// TwinCAT 3 PLC project PLC_Project
// ProgramVersion: 3.1.4024.0
// libraries:
//   Tc2_Standard, * (Beckhoff Automation GmbH)
//   Tc2_System, * (Beckhoff Automation GmbH)
//   Tc3_Module, * (Beckhoff Automation GmbH)
//   VisuDialogs, * (System)
//   VisuSymbols,3.5.10.0,System
// project tree:
//   / GlobalTextList.TcGTLO, PlcTask.TcTTO
//   GVLs/ GVL_Analogue_Transducer_Instruments.TcGVL, GVL_Analogue_Transducer_Instruments_IO_Addresses.TcGVL
//   POUs/ Analogue_Processing.TcPOU, MAIN.TcPOU
//   POUs/Function Blocks/ Sensor_Calibration_Multipoint.TcPOU, Temperature_Transducer.TcPOU
//   VISUs/ VisualizationManager.TcVMO (not stored), Visualization_Calibration_Screen.TcVIS
// real-time tasks:
//   TASK PlcTask: cycle T#10ms, priority 20, ADS port 350
// I/O:
//   DEVICE Device 1 (EtherCAT) (disabled), AmsNetId 10.0.2.15.2.1
//     Term 1 (EK1101) [EK1101 EtherCAT Coupler (2A E-Bus, ID switch)]
//       Term 2 (EL3202-0020) [EL3202-0020 2Ch. Ana. Input PT100 (RTD), High Precision, calibrated]
// variable links:
//   PLC Project/PLC Project Instance <-> Device 1 (EtherCAT)/Term 1 (EK1101)/Term 2 (EL3202-0020)
//     PlcTask Inputs/GVL_Analogue_Transducer_Instruments_IO_Addresses.Temperature_Transducer_A1_Raw_Value <-> RTD Inputs Channel 1/Value

CONFIGURATION PLC_Project
    RESOURCE PLC ON TwinCAT3
        TASK PlcTask(INTERVAL := T#10ms, PRIORITY := 20);
        PROGRAM MAIN WITH PlcTask : MAIN;
    END_RESOURCE
END_CONFIGURATION

// ---- GVLs/GVL_Analogue_Transducer_Instruments.TcGVL
//{attribute 'qualified_only'}
VAR_GLOBAL
	Temperature_Transducer_A1				:	Temperature_Transducer;
	Temperature_Transducer_A1_Calibration	:	Sensor_Calibration_Multipoint;
END_VAR

// ---- GVLs/GVL_Analogue_Transducer_Instruments_IO_Addresses.TcGVL
//	Dynamic Memory Addressing Used
//	N/B: Remember To Re-enable EtherCAT Device Under I/O If Using A Physical IPC & Intruments

VAR_GLOBAL
	Temperature_Transducer_A1_Raw_Value		AT %I*	:	INT;	//	Mapped To Term 2(EL3202-0020) Channel 1 Value
END_VAR

// ---- POUs/MAIN.TcPOU
PROGRAM MAIN
VAR
END_VAR

Analogue_Processing();

END_PROGRAM

// ---- POUs/Analogue_Processing.TcPOU
PROGRAM Analogue_Processing
VAR
END_VAR

Temperature_Transducer_A1(RawValue	:=	Temperature_Transducer_A1_Raw_Value);
Temperature_Transducer_A1_Calibration(Sensor_Input_Value := Temperature_Transducer_A1.Temperature_SI);

END_PROGRAM

// ---- POUs/Function Blocks/Temperature_Transducer.TcPOU
FUNCTION_BLOCK Temperature_Transducer
VAR_INPUT
	RawValue			:	INT			:=	0;
	SimulatedRawValue	:	INT			:=	0;
	
	InstrumentEnable	:	BOOL		:=	TRUE;
END_VAR
VAR_OUTPUT
	Temperature_SI		:	REAL		:=	0.0;			//	°C
END_VAR
VAR
	Low_Alarm			:	BOOL		:=	FALSE;
	High_Alarm			:	BOOL		:=	FALSE;
	
	Low_Alarm_Setpoint	:	REAL		:=	0.000;			//	°C
	High_Alarm_Setpoint	:	REAL		:=	100.0;			//	°C
END_VAR

IF(InstrumentEnable)THEN
	IF(SimulatedRawValue <> 0)THEN
		RawValue	:= SimulatedRawValue;
	END_IF;

	Temperature_SI		:=	INT_TO_REAL(RawValue)/ 100.0;	//	Assumes That An EL3202 16-Bit RTD IO Card Is Used To Read The PT100 Instrument

	//	Alarm Functionality: Rising Edge Required For Event System To Trigger An Alarm Event
	IF(Temperature_SI < Low_Alarm_Setpoint)THEN
		Low_Alarm		:=	TRUE;
	ELSE
		Low_Alarm		:=	FALSE;
	END_IF;

	IF(Temperature_SI > High_Alarm_Setpoint)THEN
		Low_Alarm		:=	TRUE;
	ELSE
		Low_Alarm		:=	FALSE;
	END_IF;
ELSE
	Temperature_SI		:=	0.0;
END_IF;

END_FUNCTION_BLOCK

// ---- POUs/Function Blocks/Sensor_Calibration_Multipoint.TcPOU
//	This Function Block Performs A Linear Interpolation 
//	It Uses Multiple Data Points On Which A Line Graph Can Be Plotted
//	Between Each Two Data Points, A Line Equation Exists
//	The Linear Interpolation Formula Can Then Be Used To Find A Sensor Output Value 

FUNCTION_BLOCK Sensor_Calibration_Multipoint
VAR_INPUT
	Sensor_Input_Value		:		REAL	:=	0.0;
	
	Start_Calibration		:		BOOL	:=	FALSE;
	Reset_Calibration		:		BOOL	:=	FALSE;
END_VAR
VAR_OUTPUT
	Calibrated_Output_Value	:		REAL	:=	0.0;
END_VAR
VAR	
	// Lookup Table
	Sensor_Points			:		ARRAY[1..Calibration_Points] OF REAL	:=	[0.00, 25.00, 50.00, 75.00, 100.0];		//	Sensor Input - Will Be supplied From Analogue Scaling Block
	Reference_Points		:		ARRAY[1..Calibration_Points] OF REAL	:=	[0.00, 30.55, 58.16, 69.09, 100.0];		//	Actual Value
	
	Calibration_Index		: 		UINT;
	
	//	Linear Line Equation Variables
	X1						:		REAL	:=	0.0;
	X2						:		REAL	:=	0.0;
	Y1						:		REAL	:=	0.0;
	Y2						:		REAL	:=	0.0;	
END_VAR
VAR CONSTANT
	Calibration_Points		:		UINT	:=	5;
END_VAR

FOR Calibration_Index := 1 TO Calibration_Points DO
	//	Determine Between Which Two Data Points The Sensors Value Lies
	IF(Sensor_Input_Value >= Sensor_Points[Calibration_Index] AND Sensor_Input_Value <= Sensor_Points[Calibration_Index + 1])THEN 
		//	Determine Parameters x1, x2, y1 & y2 For Straight Line Equation
		X1	:=	Sensor_Points[Calibration_Index];
		Y1	:=	Reference_Points[Calibration_Index];
		
		X2	:=	Sensor_Points[Calibration_Index + 1];
		Y2	:=	Reference_Points[Calibration_Index + 1];
		
		Calibrated_Output_Value	:= Y1 + (Sensor_Input_Value - X1)*(Y2 - Y1)/(X2 - X1);
		EXIT;
	END_IF;
END_FOR;

//	Boundary Checks
IF(Sensor_Input_Value < Sensor_Points[1])THEN
	Calibrated_Output_Value	:=	Reference_Points[1];
END_IF;

IF(Sensor_Input_Value > Sensor_Points[Calibration_Points])THEN
	Calibrated_Output_Value	:=	Reference_Points[Calibration_Points];
END_IF;

END_FUNCTION_BLOCK

// ---- GlobalTextList.TcGTLO
TEXTLIST GlobalTextList
  485 = '%32768d'
  125 = '%3d'
  748 = '%5.2f'
  165 = '%5d'
  99 = '%5f'
  587 = 'Apply Calibration'
  18 = 'Calibrated Output Value'
  547 = 'Non-Calibrated Output Value'
  655 = 'Non-Calibrated Value'
  157 = 'Raw Field Measurement'
  826 = 'Reset Calibration'
  806 = 'Sensor'
  426 = 'Sensor '
  268 = '°C'
END_TEXTLIST

// ---- VISUs/Visualization_Calibration_Screen.TcVIS
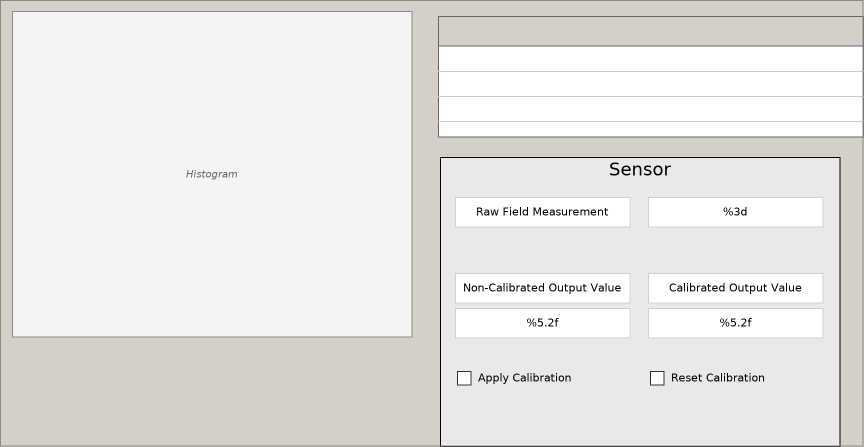
VISUALIZATION Visualization_Calibration_Screen  // 864x447
    RoundedRectangle (440,157 400x290), "Sensor"
    Histogram (12,11 400x326), scale format: %.1f, scale 0..100
        p518627256: °C
        p1518820177: Temperature_Transducer_A1_Calibration.Reference_Points
        p102497268: Temperature_Transducer_A1_Calibration.Reference_Points
        p788070771: ARRAY [1..Calibration_Points] OF REAL
    Textfield (455,308 175x30), "%5.2f", text variable: Temperature_Transducer_A1_Calibration.Sensor_Input_Value
    Textfield (455,273 175x30), "Non-Calibrated Output Value"
    Table (438,16 426x121), data array: Temperature_Transducer_A1_Calibration.Reference_Points
        p3854506369: Temperature_Transducer_A1_Calibration.Reference_Points[INDEX]
    Textfield (648,308 175x30), "%5.2f", text variable: Temperature_Transducer_A1_Calibration.Calibrated_Output_Value
    Textfield (648,273 175x30), "Calibrated Output Value"
    Checkbox (455,363 150x30), "Apply Calibration", variable: Temperature_Transducer_A1_Calibration.Start_Calibration
    Checkbox (648,363 150x30), "Reset Calibration", variable: Temperature_Transducer_A1_Calibration.Reset_Calibration
    Textfield (455,197 175x30), "Raw Field Measurement"
    Textfield (648,197 175x30), "%3d", text variable: Temperature_Transducer_A1.SimulatedRawValue
        OnMouseDown: write the text variable via Default, min 0, max 32768
END_VISUALIZATION
